// TIA Portal V17 export
// export: Created 2024-09-02T12:50:25.4947099Z, ExportSetting WithDefaults, DisplayName Totally Integrated Automation Portal, DisplayVersion V17, DisplayName TIA Portal Openness, DisplayVersion V17, DisplayName TIA Portal Version Control Interface, DisplayVersion V17, DisplayName STEP 7 Professional, DisplayVersion V17, DisplayName STEP 7 Safety, DisplayVersion V17, DisplayName WinCC Professional, DisplayVersion V17
VAR_GLOBAL   // PLC tag table "MES_Constant"
END_VAR
VAR_GLOBAL CONSTANT   // user constants
   Comunication_MES_Init_Step : Int := 0;
   Comunication_MES_Ready : Int := 2;
   Comunication_MES_Finished_OK : Int := 3;
   Status_Of_Pallet_OK_MES : Int := 1;
   Status_Of_Pallet_Autorization_OK : Int := 1;
   Comunication_PLC_Ready : Int := 1;
   Comunication_MES_Finished_NOK : Int := 4;
END_VAR
